Staubli VAL3: S7telegram_T.pjx

Parameters version=s7.9.1 stackSize=5000 millimeterUnit=true
Data file=S7telegram_T.dtx
